FUNCTION_BLOCK FB_TDS323PC57 EXTENDS FB_ModbusSlave
VAR
	arrConditionData	:	ARRAY [0..31] OF REAL;
	arrUp_LoLimit		:	ARRAY [0..31] OF REAL;
	arrUpUp_UpLimit		:	ARRAY [0..31] OF REAL;
END_VAR

PROPERTY ConditionData : ARRAY [0..31] OF REAL
GET
ConditionData := arrConditionData;
END_GET
END_PROPERTY

METHOD Convert : BOOL
VAR_INPUT
	iRegionNo	:	INT;
	pReadData	:	POINTER TO BYTE;
END_VAR
VAR
	pTempData	: 	POINTER TO BYTE;
	iTempData	: 	BYTE;
	iLoop		: 	INT;
	bHiByte		:	BOOL := TRUE;
	iLoopStart	:	INT;
	iLoopEnd	:	INT;
	arrTempData	:	ARRAY [0..8] OF WORD;
END_VAR
FOR iLoop := 0 TO 7 DO
	arrTempData[iLoop] := SHL(BYTE_TO_WORD(pReadData[iLoop*2+3]), 8);
	arrTempData[iLoop] := arrTempData[iLoop] + BYTE_TO_WORD(pReadData[iLoop*2+3+1]);
	IF bSwap THEN
		arrTempData[iLoop] := ROL(arrTempData[iLoop], 8);
	END_IF
END_FOR

CASE iRegionNo OF 
	0: 
		iLoopStart := 0;
		iLoopEnd := 7;
		
	1: 
		iLoopStart := 8;
		iLoopEnd := 15;
		
	2: 
		iLoopStart := 16;
		iLoopEnd := 23;

	3: 
		iLoopStart := 24;
		iLoopEnd := 31;
	
END_CASE

FOR iLoop := 0 TO 7 DO 
	arrConditionData[iLoopStart + iLoop] := WORD_TO_REAL(arrTempData[iLoop]);
END_FOR
END_METHOD

METHOD FirstCycle : BOOL
VAR_INPUT
END_VAR
arrAddress[0][0] := 16#0000;
arrAddress[0][1] := 8;
arrAddress[1][0] := 16#0008;
arrAddress[1][1] := 8;
arrAddress[2][0] := 16#0010;
arrAddress[2][1] := 8;
arrAddress[3][0] := 16#0018;
arrAddress[3][1] := 8;

iNumAddRegion := 4;

bSwap := FALSE;
END_METHOD

PROPERTY Up_LoLimit : ARRAY [0..63] OF WORD
GET
Up_LoLimit := arrUp_LoLimit;
END_GET
END_PROPERTY

PROPERTY UpUp_UpLimit : ARRAY [0..63] OF WORD
GET
UpUp_UpLimit := arrUpUp_UpLimit;
END_GET
END_PROPERTY

END_FUNCTION_BLOCK

(* stored: Version 1.1.0.1, ProductVersion 3.1.4024.12
   POU FB_TDS323PC57: Id {e8fb70df-be29-4460-957f-9586549f42be}, SpecialFunc None
   Property ConditionData: Id {f85b153e-777c-46bf-afd8-d7a098fe9e2d}
   Get Get: Id {a26145bd-6d63-412a-ae13-c34a1165bf75}
   Method Convert: Id {b48e17b2-54ba-4775-8ece-9ac9c943983a}
   Method FirstCycle: Id {70eeedf9-dc8a-4bd4-9ac7-1fc925a31989}
   Property Up_LoLimit: Id {d5b8ab1e-d642-46de-8c6b-98e1a26d2cb6}
   Get Get: Id {e20bdbc2-bf8e-4486-913d-26f0a21b8c5f}
   Property UpUp_UpLimit: Id {c107981f-2291-4349-8d24-74209dc61e7b}
   Get Get: Id {6abb6c8a-f004-493f-b539-3cad41bef48c} *)
